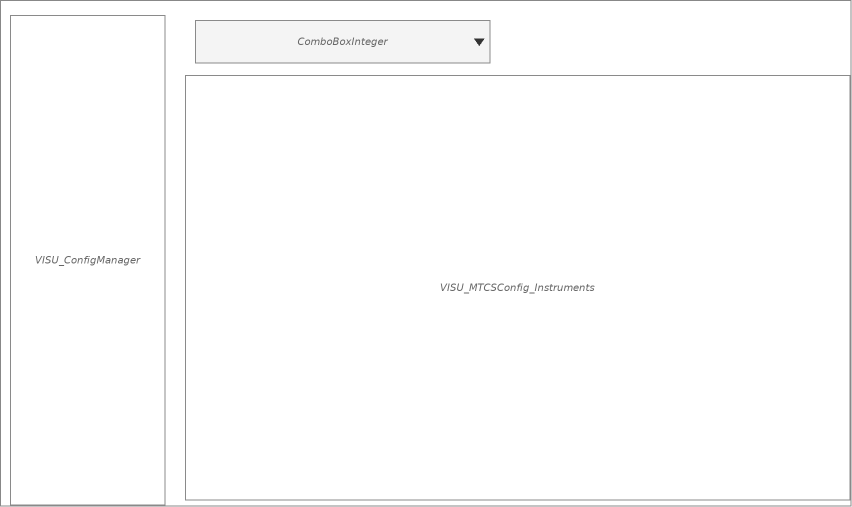
VISUALIZATION VISU_MTCSConfig  // 852x507
VAR_IN_OUT
    editableConfig : MTCSConfig;
	activeConfig : MTCSConfig;
    mgr : ConfigManager;
    mgrWidget : ConfigManagerWidget;
    widget : MTCSWidget;
END_VAR
    ComboBoxInteger (195,20 295x43), variable: widget.configActiveTab, text list: 'MTCSConfigTabsTextList'
    Frame (185,75 665x425), frame switch variable: widget.configActiveTab
        shows VISU_MTCSConfig_Instruments(active := activeConfig.instruments, editable := editableConfig.instruments, currentPosition := widget.configInstrumentsActiveTab)
        shows VISU_MTCSConfig_Location(active := activeConfig.location, editable := editableConfig.location)
    Frame (10,15 155x490)
        shows VISU_ConfigManager(mgr := mgr, widget := mgrWidget)
END_VISUALIZATION

(* stored: Version 1.1.0.1, ProductVersion 3.1.4019.2
   Visu VISU_MTCSConfig: Id {675cfe03-28f2-4d9e-968a-a8b0ae8ca3c8} *)
